{attribute 'qualified_only'}
{attribute 'strict'}
TYPE E_CNC_Robot_Command :
(
	NoCommand 						:= 0,
	Home							:= 1,
	QuickHome						:= 2,
	Wait							:= 3,
	Service							:= 4,
	Pick_Up_CNC 					:= 5,
	Put_Down_CNC					:= 6,
	Pick_Up_Lifter	 				:= 7,
	Put_Down_Lifter 				:= 8,
	Camera_Lifter					:= 9,
	Pick_Up_Master 					:= 10,
	Put_Down_Master					:= 11,
	Pick_Up_Master_From_Lifter		:= 12,
	Put_Down_Master_To_Lifter		:= 13
);
END_TYPE

(* stored: Version 1.1.0.1, ProductVersion 3.1.4024.12
   DUT E_CNC_Robot_Command: Id {a652049e-e2eb-4a3a-83c9-13e0156f2241} *)
